NETWORK
TITLE =ML_LABORFREIGABE_T6
// Act 031
// Box           : LT-CIP
// Output address: Q258.5
      CALL FC    70 (
           UnitNo                   := #UnitNo,
           ActRec                   := DB2060.ML_LABORFREIGABE_T6,
           Typ                      := 0,
           FBa                      := #xTmp,
           FBa2                     := #xTmp,
           Out                      := Q    258.5);

END_FUNCTION_BLOCK

FUNCTION_BLOCK FB 1061
TITLE =U006: Water Tank 6
FAMILY : BOTEC_F1
NAME : UniE
VERSION : 1.2


VAR_TEMP
  CIP : BOOL ;	//CIP active
  UNIM : BOOL ;	//Unit Not In Maintenance
  GenRel : BOOL ;	//general OK (emergency and maintenance OK)
  EStopOK : BOOL ;	//emergency OK
  UnitNo : INT ;	//unit number
  xTmp : BOOL ;	//Temporary Bool
  iTmp : INT ;	//Temporary INT
  rTmp : REAL ;	//Temporary REAL
  dTmp : DINT ;	//Temporary DINT (free for general use)
  RetValInt : INT ;	//return value
END_VAR
BEGIN
NETWORK
TITLE =General

      SET   ;
// Simulation ---------------------------------------------------------------
      A     DB1061.DBX 1357.7;
      CC    FB  1069; // "WT06Sim"
      A     DB1061.DBX   17.3;
      =     DB1061.DBX 1357.7; //Help bit for simulation

// get unit number ----------------------------------------------------------
      L     DB1060.DBW    0;
      T     #UnitNo;

// communication ------------------------------------------------------------
      UC    FB  1065; // WT06Com

NETWORK
TITLE =Sequence organisation

      CLR   ;
      =     M    122.2;

// CIP Counter
      CALL FC    29 (
           UnitNo                   := #UnitNo,
           Value                    := DB1065.DBD   54,
           Enable                   := TRUE,
           Down                     := FALSE,
           OriginDetect             := 0.000000e+000,
           MaxDiffPS                := 1.000000e+000,
           SFMRec                   := DB1061.Seq.SFM[15],
           ValueOld                 := DB1061.DBD 1418);

// sequencer ----------------------------------------------------------------
      A     DB1063.DBX   43.1;
      S     DB1063.DBX   97.3;

      CALL FC    40 (
           UnitNo                   := #UnitNo);

END_FUNCTION_BLOCK

FUNCTION_BLOCK FB 1070
TITLE =U007: Wassertank 07
FAMILY : BOTEC_F1
NAME : U007A
VERSION : 2.1


VAR_TEMP
  EStopOK : BOOL ;	//auxiliary flag
  CIP : BOOL ;	//CIP Program Selected
  xTmp : BOOL ;	//Temporary Bool(free for general use)
  DummyBool : BOOL ;	//Temporary Bool(free for general use)
  UnitNo : INT ;	//unit number
  UnitFB : INT ;	//unit expansion FB number
  rTmp : REAL ;	//Temporary REAL (free for general use)
  iTmp : INT ;	//Temporary INT (free for general use)
  DummyInt : INT ;	//Temporary INT (free for general use)
  dTmp : DINT ;	//Temporary DINT (free for general use)
END_VAR
BEGIN
NETWORK
TITLE =general

      CLR   ;
      =     #xTmp;
      =     #EStopOK;

      L     DB1070.DBW    0;
      T     #UnitNo;
      L     DB1070.DBW    2;
      T     #UnitFB;

NETWORK
TITLE =analog inputs

      NOP   0;
// LI_T7 AnI 001 Inhalt Tank 7
      CALL FC    24 (
           UnitNo                   := #UnitNo,
           AnIRec                   := DB2073.LI_T7,
           ValPer                   := DB302.DBW   76);

NETWORK
TITLE =Universal value

      NOP   0;
// unv001 UnV 001 Process Status
      CALL FC    27 (
           UnitNo                   := #UnitNo,
           UnVRec                   := DB2075.unv001,
           ValExt                   := DB2075.DBD  234);

// unv002 UnV 002 Universal Value 02
      CALL FC    27 (
           UnitNo                   := #UnitNo,
           UnVRec                   := DB2075.unv002,
           ValExt                   := DB2075.DBD  362);

// unv003 UnV 003 Universal Value 03
      CALL FC    27 (
           UnitNo                   := #UnitNo,
           UnVRec                   := DB2075.unv003,
           ValExt                   := DB2075.DBD  490);

NETWORK
TITLE =special inputs

      NOP   0;
// LS_LLL_T7 SpI 001
      CALL FC    14 (
           UnitNo                   := #UnitNo,
           SpIRec                   := DB2071.LS_LLL_T7,
           SpIBit                   := I     71.0);

// LS_HL_T7 SpI 002
      CALL FC    14 (
           UnitNo                   := #UnitNo,
           SpIRec                   := DB2071.LS_HL_T7,
           SpIBit                   := I     70.6);

// LS_LL_T7 SpI 005
      CALL FC    14 (
           UnitNo                   := #UnitNo,
           SpIRec                   := DB2071.LS_LL_T7,
           SpIBit                   := I     70.7);

// RM_NI_T7_K2 SpI 008
      CALL FC    14 (
           UnitNo                   := #UnitNo,
           SpIRec                   := DB2071.RM_NI_T7_K2,
           SpIBit                   := I     61.2);

// RM_NI_T7_K3 SpI 010
      CALL FC    14 (
           UnitNo                   := #UnitNo,
           SpIRec                   := DB2071.RM_NI_T7_K3,
           SpIBit                   := I     69.4);

// LABOR_FREIG_T7 SpI 011 SCHLUESSELSCHALTER LABOR
      CALL FC    14 (
           UnitNo                   := #UnitNo,
           SpIRec                   := DB2071.LABOR_FREIG_T7,
           SpIBit                   := I    258.6);

NETWORK
TITLE =messages

      NOP   0;
// msg001 Msg 001 Message 01
      CALL FC    16 (
           UnitNo                   := #UnitNo,
           MsgRec                   := DB2077.msg001,
           MsgBit                   := DB2077.DBX   82.7);

// msg002 Msg 002 Message 02
      CALL FC    16 (
           UnitNo                   := #UnitNo,
           MsgRec                   := DB2077.msg002,
           MsgBit                   := DB2077.DBX  142.7);

NETWORK
TITLE =unit supply

      UC    FB [#UnitFB];

NETWORK
TITLE =T7_FW
// Act 001
// Box           : Ventilinsel 5
// Input address : I338.3
// Output address: Q338.3
      CALL FC    70 (
           UnitNo                   := #UnitNo,
           ActRec                   := DB2070.T7_FW,
           Typ                      := 1,
           FBa                      := #xTmp,
           FBa2                     := I    338.3,
           Out                      := Q    338.3);

NETWORK
TITLE =T7_KEG
// Act 003
// Box           : Ventilinsel 5
// Input address : I339.1
// Output address: Q339.1
      CALL FC    70 (
           UnitNo                   := #UnitNo,
           ActRec                   := DB2070.T7_KEG,
           Typ                      := 1,
           FBa                      := #xTmp,
           FBa2                     := I    339.1,
           Out                      := Q    339.1);

NETWORK
TITLE =T7_SK
// Act 004
// Box           : Ventilinsel 5
// Input address : I338.0
// Output address: Q338.0
      CALL FC    70 (
           UnitNo                   := #UnitNo,
           ActRec                   := DB2070.T7_SK,
           Typ                      := 1,
           FBa                      := #xTmp,
           FBa2                     := I    338.0,
           Out                      := Q    338.0);

NETWORK
TITLE =T7_A10
// Act 005
// Box           : Ventilinsel 2
// Input address : I316.2
// Output address: Q316.2
      CALL FC    70 (
           UnitNo                   := #UnitNo,
           ActRec                   := DB2070.T7_A10,
           Typ                      := 1,
           FBa                      := #xTmp,
           FBa2                     := I    316.2,
           Out                      := Q    316.2);

NETWORK
TITLE =T7_A9
// Act 006
// Box           : Ventilinsel 2
// Input address : I318.2
// Output address: Q318.2
      CALL FC    70 (
           UnitNo                   := #UnitNo,
           ActRec                   := DB2070.T7_A9,
           Typ                      := 1,
           FBa                      := #xTmp,
           FBa2                     := I    318.2,
           Out                      := Q    318.2);

NETWORK
TITLE =T7_A12
// Act 007
// Box           : Ventilinsel 2
// Input address : I320.2
// Output address: Q320.2
      CALL FC    70 (
           UnitNo                   := #UnitNo,
           ActRec                   := DB2070.T7_A12,
           Typ                      := 1,
           FBa                      := #xTmp,
           FBa2                     := I    320.2,
           Out                      := Q    320.2);

NETWORK
TITLE =T7_A7
// Act 008
// Box           : Ventilinsel 2
// Input address : I322.2
// Output address: Q322.2
      CALL FC    70 (
           UnitNo                   := #UnitNo,
           ActRec                   := DB2070.T7_A7,
           Typ                      := 1,
           FBa                      := #xTmp,
           FBa2                     := I    322.2,
           Out                      := Q    322.2);

NETWORK
TITLE =T7_A8
// Act 009
// Box           : Ventilinsel 3
// Input address : I324.2
// Output address: Q324.2
      CALL FC    70 (
           UnitNo                   := #UnitNo,
           ActRec                   := DB2070.T7_A8,
           Typ                      := 1,
           FBa                      := #xTmp,
           FBa2                     := I    324.2,
           Out                      := Q    324.2);

NETWORK
TITLE =T7_A5
// Act 010
// Box           : Ventilinsel 3
// Input address : I326.2
// Output address: Q326.2
      CALL FC    70 (
           UnitNo                   := #UnitNo,
           ActRec                   := DB2070.T7_A5,
           Typ                      := 1,
           FBa                      := #xTmp,
           FBa2                     := I    326.2,
           Out                      := Q    326.2);

NETWORK
TITLE =T7_A11
// Act 011
// Box           : Ventilinsel 3
// Input address : I328.2
// Output address: Q328.2
      CALL FC    70 (
           UnitNo                   := #UnitNo,
           ActRec                   := DB2070.T7_A11,
           Typ                      := 1,
           FBa                      := #xTmp,
           FBa2                     := I    328.2,
           Out                      := Q    328.2);

NETWORK
TITLE =T7_A14
// Act 012
// Box           : Ventilinsel 4
// Input address : I330.2
// Output address: Q330.2
      CALL FC    70 (
           UnitNo                   := #UnitNo,
           ActRec                   := DB2070.T7_A14,
           Typ                      := 1,
           FBa                      := #xTmp,
           FBa2                     := I    330.2,
           Out                      := Q    330.2);

NETWORK
TITLE =T7_A15
// Act 013
// Box           : Ventilinsel 4
// Input address : I332.2
// Output address: Q332.2
      CALL FC    70 (
           UnitNo                   := #UnitNo,
           ActRec                   := DB2070.T7_A15,
           Typ                      := 0,
           FBa                      := #xTmp,
           FBa2                     := I    332.2,
           Out                      := Q    332.2);

NETWORK
TITLE =T7_RR1
// Act 014
// Box           : Ventilinsel 4
// Input address : I334.2
// Output address: Q334.2
      CALL FC    70 (
           UnitNo                   := #UnitNo,
           ActRec                   := DB2070.T7_RR1,
           Typ                      := 1,
           FBa                      := #xTmp,
           FBa2                     := I    334.2,
           Out                      := Q    334.2);

NETWORK
TITLE =RV1_T7  RV1_T7 Ventil CIP Vorlauf Tank 7
// Act 015
// Box           : VS2-BB
// Input address : I304.1
// Output address: Q304.1
      CALL FC    70 (
           UnitNo                   := #UnitNo,
           ActRec                   := DB2070.RV1_T7,
           Typ                      := 1,
           FBa                      := #xTmp,
           FBa2                     := I    304.1,
           Out                      := Q    304.1);

NETWORK
TITLE =B6F_T7  B6F_T7
// Act 016
// Box           : VS2-BB
// Input address : I304.5
// Output address: Q304.5
      CALL FC    70 (
           UnitNo                   := #UnitNo,
           ActRec                   := DB2070.B6F_T7,
           Typ                      := 1,
           FBa                      := #xTmp,
           FBa2                     := I    304.5,
           Out                      := Q    304.5);

NETWORK
TITLE =H6F_T7  H6F_T7
// Act 017
// Box           : VS2-BB
// Input address : I304.4
// Output address: Q304.4
      CALL FC    70 (
           UnitNo                   := #UnitNo,
           ActRec                   := DB2070.H6F_T7,
           Typ                      := 1,
           FBa                      := #xTmp,
           FBa2                     := I    304.4,
           Out                      := Q    304.4);

NETWORK
TITLE =J6F_T7  J6F_T7
// Act 018
// Box           : VS2-BB
// Input address : I304.6
// Output address: Q304.6
      CALL FC    70 (
           UnitNo                   := #UnitNo,
           ActRec                   := DB2070.J6F_T7,
           Typ                      := 1,
           FBa                      := #xTmp,
           FBa2                     := I    304.6,
           Out                      := Q    304.6);

NETWORK
TITLE =L6F_T7  L6F_T7
// Act 019
// Box           : VS2-BB
// Input address : I304.7
// Output address: Q304.7
      CALL FC    70 (
           UnitNo                   := #UnitNo,
           ActRec                   := DB2070.L6F_T7,
           Typ                      := 1,
           FBa                      := #xTmp,
           FBa2                     := I    304.7,
           Out                      := Q    304.7);

NETWORK
TITLE =D6_T7  D6_T7
// Act 020
// Box           : VS2-BB
// Input address : I305.1
// Output address: Q305.1
      CALL FC    70 (
           UnitNo                   := #UnitNo,
           ActRec                   := DB2070.D6_T7,
           Typ                      := 1,
           FBa                      := #xTmp,
           FBa2                     := I    305.1,
           Out                      := Q    305.1);

NETWORK
TITLE =B6_T7  B6_T7
// Act 021
// Box           : VS2-BB
// Input address : I305.0
// Output address: Q305.0
      CALL FC    70 (
           UnitNo                   := #UnitNo,
           ActRec                   := DB2070.B6_T7,
           Typ                      := 1,
           FBa                      := #xTmp,
           FBa2                     := I    305.0,
           Out                      := Q    305.0);

NETWORK
TITLE =A_T7  A_T7
// Act 022
// Box           : VS2-BB
// Input address : I304.2
// Output address: Q304.2
      CALL FC    70 (
           UnitNo                   := #UnitNo,
           ActRec                   := DB2070.A_T7,
           Typ                      := 1,
           FBa                      := #xTmp,
           FBa2                     := I    304.2,
           Out                      := Q    304.2);

NETWORK
TITLE =B_T7  B_T7
// Act 023
// Box           : VS2-BB
// Input address : I304.3
// Output address: Q304.3
      CALL FC    70 (
           UnitNo                   := #UnitNo,
           ActRec                   := DB2070.B_T7,
           Typ                      := 1,
           FBa                      := #xTmp,
           FBa2                     := I    304.3,
           Out                      := Q    304.3);

NETWORK
TITLE =CF_T7
// Act 024
// Box           : Ventilinsel 1
// Input address : I17.0
// Output address: Q17.0
      CALL FC    70 (
           UnitNo                   := #UnitNo,
           ActRec                   := DB2070.CF_T7,
           Typ                      := 1,
           FBa                      := #xTmp,
           FBa2                     := I     17.0,
           Out                      := Q     17.0);

NETWORK
TITLE =RW5_T7  RW5_T7
// Act 026
// Box           : VS2-BB
// Input address : I305.2
// Output address: Q305.2
      CALL FC    70 (
           UnitNo                   := #UnitNo,
           ActRec                   := DB2070.RW5_T7,
           Typ                      := 1,
           FBa                      := #xTmp,
           FBa2                     := I    305.2,
           Out                      := Q    305.2);

NETWORK
TITLE =RW6_T7  RW6_T7
// Act 027
// Box           : VS2-BB
// Input address : I305.3
// Output address: Q305.3
      CALL FC    70 (
           UnitNo                   := #UnitNo,
           ActRec                   := DB2070.RW6_T7,
           Typ                      := 1,
           FBa                      := #xTmp,
           FBa2                     := I    305.3,
           Out                      := Q    305.3);

NETWORK
TITLE =VR_T7  VR_T7
// Act 029
// Box           : VS2-BB
// Output address: Q305.4
      CALL FC    70 (
           UnitNo                   := #UnitNo,
           ActRec                   := DB2070.VR_T7,
           Typ                      := 0,
           FBa                      := #xTmp,
           FBa2                     := #xTmp,
           Out                      := Q    305.4);

NETWORK
TITLE =ML_LABORFREIGABE_T7
// Act 031
// Box           : LT-CIP
// Output address: Q258.6
      CALL FC    70 (
           UnitNo                   := #UnitNo,
           ActRec                   := DB2070.ML_LABORFREIGABE_T7,
           Typ                      := 0,
           FBa                      := #xTmp,
           FBa2                     := #xTmp,
           Out                      := Q    258.6);

END_FUNCTION_BLOCK

FUNCTION_BLOCK FB 1071
TITLE =U007: Water Tank 7
FAMILY : BOTEC_F1
NAME : UniE
VERSION : 1.2


VAR_TEMP
  CIP : BOOL ;	//CIP active
  UNIM : BOOL ;	//Unit Not In Maintenance
  GenRel : BOOL ;	//general OK (emergency and maintenance OK)
  EStopOK : BOOL ;	//emergency OK
  UnitNo : INT ;	//unit number
  xTmp : BOOL ;	//Temporary Bool
  iTmp : INT ;	//Temporary INT
  rTmp : REAL ;	//Temporary REAL
  dTmp : DINT ;	//Temporary DINT (free for general use)
  RetValInt : INT ;	//return value
END_VAR
BEGIN
NETWORK
TITLE =General

      SET   ;
// Simulation ---------------------------------------------------------------
      A     DB1071.DBX 1357.7;
      CC    FB  1079; // "WT07Sim"
      A     DB1071.DBX   17.3;
      =     DB1071.DBX 1357.7; //Help bit for simulation

// get unit number ----------------------------------------------------------
      L     DB1070.DBW    0;
      T     #UnitNo;


// communication ------------------------------------------------------------
      UC    FB  1075; // WT07Com

NETWORK
TITLE =Sequence organisation

      CLR   ;
      =     M    122.2;

// CIP Counter
      CALL FC    29 (
           UnitNo                   := #UnitNo,
           Value                    := DB1075.DBD   54,
           Enable                   := TRUE,
           Down                     := FALSE,
           OriginDetect             := 0.000000e+000,
           MaxDiffPS                := 1.000000e+000,
           SFMRec                   := DB1071.Seq.SFM[15],
           ValueOld                 := DB1071.DBD 1418);

// sequencer ----------------------------------------------------------------
      A     DB1073.DBX   43.1;
      S     DB1073.DBX   97.3;

      CALL FC    40 (
           UnitNo                   := #UnitNo);

END_FUNCTION_BLOCK

FUNCTION_BLOCK FB 1080
TITLE =U008: Wassertank 08
FAMILY : BOTEC_F1
NAME : U008A
VERSION : 2.1


VAR_TEMP
  EStopOK : BOOL ;	//auxiliary flag
  CIP : BOOL ;	//CIP Program Selected
  xTmp : BOOL ;	//Temporary Bool(free for general use)
  DummyBool : BOOL ;	//Temporary Bool(free for general use)
  UnitNo : INT ;	//unit number
  UnitFB : INT ;	//unit expansion FB number
  rTmp : REAL ;	//Temporary REAL (free for general use)
  iTmp : INT ;	//Temporary INT (free for general use)
  DummyInt : INT ;	//Temporary INT (free for general use)
  dTmp : DINT ;	//Temporary DINT (free for general use)
END_VAR
BEGIN
NETWORK
TITLE =general

      CLR   ;
      =     #xTmp;
      =     #EStopOK;

      L     DB1080.DBW    0;
      T     #UnitNo;
      L     DB1080.DBW    2;
      T     #UnitFB;

NETWORK
TITLE =analog inputs

      NOP   0;
// LI_T8 AnI 001 Inhalt Tank 8
      CALL FC    24 (
           UnitNo                   := #UnitNo,
           AnIRec                   := DB2083.LI_T8,
           ValPer                   := DB302.DBW   78);

NETWORK
TITLE =Universal value

      NOP   0;
// unv001 UnV 001 Process Status
      CALL FC    27 (
           UnitNo                   := #UnitNo,
           UnVRec                   := DB2085.unv001,
           ValExt                   := DB2085.DBD  234);

// unv002 UnV 002 Universal Value 02
      CALL FC    27 (
           UnitNo                   := #UnitNo,
           UnVRec                   := DB2085.unv002,
           ValExt                   := DB2085.DBD  362);

// unv003 UnV 003 Universal Value 03
      CALL FC    27 (
           UnitNo                   := #UnitNo,
           UnVRec                   := DB2085.unv003,
           ValExt                   := DB2085.DBD  490);

NETWORK
TITLE =special inputs

      NOP   0;
// LS_LLL_T8 SpI 001
      CALL FC    14 (
           UnitNo                   := #UnitNo,
           SpIRec                   := DB2081.LS_LLL_T8,
           SpIBit                   := I    184.7);

// LS_HL_T8 SpI 002
      CALL FC    14 (
           UnitNo                   := #UnitNo,
           SpIRec                   := DB2081.LS_HL_T8,
           SpIBit                   := I    184.5);

// RM_NI_T8_ML SpI 003
      CALL FC    14 (
           UnitNo                   := #UnitNo,
           SpIRec                   := DB2081.RM_NI_T8_ML,
           SpIBit                   := I    184.4);

// RM_NI_T8_VV SpI 004 RM Vacuumventil Tank 8 ZU=1
      CALL FC    14 (
           UnitNo                   := #UnitNo,
           SpIRec                   := DB2081.RM_NI_T8_VV,
           SpIBit                   := I    184.6);

// LS_LL_T8 SpI 005
      CALL FC    14 (
           UnitNo                   := #UnitNo,
           SpIRec                   := DB2081.LS_LL_T8,
           SpIBit                   := I    185.7);

// RM_NI_T8_K4_AUF SpI 006 RM Klappe vor Filter Tank 8 AUF=1
      CALL FC    14 (
           UnitNo                   := #UnitNo,
           SpIRec                   := DB2081.RM_NI_T8_K4_AUF,
           SpIBit                   := I    186.1);

// RM_NI_T8_K4_ZU SpI 007 RM Klappe vor Filter Tank 8 ZU=1
      CALL FC    14 (
           UnitNo                   := #UnitNo,
           SpIRec                   := DB2081.RM_NI_T8_K4_ZU,
           SpIBit                   := I    184.3);

// RM_NI_T8_K2 SpI 008
      CALL FC    14 (
           UnitNo                   := #UnitNo,
           SpIRec                   := DB2081.RM_NI_T8_K2,
           SpIBit                   := I    184.1);

// RM_NI_T8_K3 SpI 010
      CALL FC    14 (
           UnitNo                   := #UnitNo,
           SpIRec                   := DB2081.RM_NI_T8_K3,
           SpIBit                   := I    184.2);

// LABOR_FREIG_T8 SpI 011 SCHLUESSELSCHALTER LABOR
      CALL FC    14 (
           UnitNo                   := #UnitNo,
           SpIRec                   := DB2081.LABOR_FREIG_T8,
           SpIBit                   := I    259.0);

NETWORK
TITLE =messages

      NOP   0;
// msg001 Msg 001 Message 01
      CALL FC    16 (
           UnitNo                   := #UnitNo,
           MsgRec                   := DB2087.msg001,
           MsgBit                   := DB2087.DBX   82.7);

// msg002 Msg 002 Message 02
      CALL FC    16 (
           UnitNo                   := #UnitNo,
           MsgRec                   := DB2087.msg002,
           MsgBit                   := DB2087.DBX  142.7);

NETWORK
TITLE =unit supply

      UC    FB [#UnitFB];

NETWORK
TITLE =T8_A10
// Act 005
// Box           : Ventilinsel 2
// Input address : I316.1
// Output address: Q316.1
      CALL FC    70 (
           UnitNo                   := #UnitNo,
           ActRec                   := DB2080.T8_A10,
           Typ                      := 1,
           FBa                      := #xTmp,
           FBa2                     := I    316.1,
           Out                      := Q    316.1);

NETWORK
TITLE =T8_A9
// Act 006
// Box           : Ventilinsel 2
// Input address : I318.1
// Output address: Q318.1
      CALL FC    70 (
           UnitNo                   := #UnitNo,
           ActRec                   := DB2080.T8_A9,
           Typ                      := 1,
           FBa                      := #xTmp,
           FBa2                     := I    318.1,
           Out                      := Q    318.1);

NETWORK
TITLE =T8_A12
// Act 007
// Box           : Ventilinsel 2
// Input address : I320.1
// Output address: Q320.1
      CALL FC    70 (
           UnitNo                   := #UnitNo,
           ActRec                   := DB2080.T8_A12,
           Typ                      := 1,
           FBa                      := #xTmp,
           FBa2                     := I    320.1,
           Out                      := Q    320.1);

NETWORK
TITLE =T8_A7
// Act 008
// Box           : Ventilinsel 2
// Input address : I322.1
// Output address: Q322.1
      CALL FC    70 (
           UnitNo                   := #UnitNo,
           ActRec                   := DB2080.T8_A7,
           Typ                      := 1,
           FBa                      := #xTmp,
           FBa2                     := I    322.1,
           Out                      := Q    322.1);

NETWORK
TITLE =T8_A8
// Act 009
// Box           : Ventilinsel 3
// Input address : I324.1
// Output address: Q324.1
      CALL FC    70 (
           UnitNo                   := #UnitNo,
           ActRec                   := DB2080.T8_A8,
           Typ                      := 1,
           FBa                      := #xTmp,
           FBa2                     := I    324.1,
           Out                      := Q    324.1);

NETWORK
TITLE =T8_A5
// Act 010
// Box           : Ventilinsel 3
// Input address : I326.1
// Output address: Q326.1
      CALL FC    70 (
           UnitNo                   := #UnitNo,
           ActRec                   := DB2080.T8_A5,
           Typ                      := 1,
           FBa                      := #xTmp,
           FBa2                     := I    326.1,
           Out                      := Q    326.1);

NETWORK
TITLE =T8_A11
// Act 011
// Box           : Ventilinsel 3
// Input address : I328.1
// Output address: Q328.1
      CALL FC    70 (
           UnitNo                   := #UnitNo,
           ActRec                   := DB2080.T8_A11,
           Typ                      := 1,
           FBa                      := #xTmp,
           FBa2                     := I    328.1,
           Out                      := Q    328.1);

NETWORK
TITLE =T8_A14
// Act 012
// Box           : Ventilinsel 4
// Input address : I330.1
// Output address: Q330.1
      CALL FC    70 (
           UnitNo                   := #UnitNo,
           ActRec                   := DB2080.T8_A14,
           Typ                      := 1,
           FBa                      := #xTmp,
           FBa2                     := I    330.1,
           Out                      := Q    330.1);

NETWORK
TITLE =T8_A15
// Act 013
// Box           : Ventilinsel 4
// Input address : I332.1
// Output address: Q332.1
      CALL FC    70 (
           UnitNo                   := #UnitNo,
           ActRec                   := DB2080.T8_A15,
           Typ                      := 0,
           FBa                      := #xTmp,
           FBa2                     := I    332.1,
           Out                      := Q    332.1);

NETWORK
TITLE =T8_RR1
// Act 014
// Box           : Ventilinsel 4
// Input address : I334.1
// Output address: Q334.1
      CALL FC    70 (
           UnitNo                   := #UnitNo,
           ActRec                   := DB2080.T8_RR1,
           Typ                      := 1,
           FBa                      := #xTmp,
           FBa2                     := I    334.1,
           Out                      := Q    334.1);

NETWORK
TITLE =RV1_T8  RV1_T8
// Act 015
// Box           : VS2-BB
// Input address : I305.5
// Output address: Q305.5
      CALL FC    70 (
           UnitNo                   := #UnitNo,
           ActRec                   := DB2080.RV1_T8,
           Typ                      := 1,
           FBa                      := #xTmp,
           FBa2                     := I    305.5,
           Out                      := Q    305.5);

NETWORK
TITLE =B6F_T8  B6F_T8
// Act 016
// Box           : VS2-BB
// Input address : I306.1
// Output address: Q306.1
      CALL FC    70 (
           UnitNo                   := #UnitNo,
           ActRec                   := DB2080.B6F_T8,
           Typ                      := 1,
           FBa                      := #xTmp,
           FBa2                     := I    306.1,
           Out                      := Q    306.1);

NETWORK
TITLE =H6F_T8  H6F_T8
// Act 017
// Box           : VS2-BB
// Input address : I306.0
// Output address: Q306.0
      CALL FC    70 (
           UnitNo                   := #UnitNo,
           ActRec                   := DB2080.H6F_T8,
           Typ                      := 1,
           FBa                      := #xTmp,
           FBa2                     := I    306.0,
           Out                      := Q    306.0);

NETWORK
TITLE =J6F_T8  J6F_T8
// Act 018
// Box           : VS2-BB
// Input address : I306.2
// Output address: Q306.2
      CALL FC    70 (
           UnitNo                   := #UnitNo,
           ActRec                   := DB2080.J6F_T8,
           Typ                      := 1,
           FBa                      := #xTmp,
           FBa2                     := I    306.2,
           Out                      := Q    306.2);

NETWORK
TITLE =L6F_T8  L6F_T8
// Act 019
// Box           : VS2-BB
// Input address : I306.3
// Output address: Q306.3
      CALL FC    70 (
           UnitNo                   := #UnitNo,
           ActRec                   := DB2080.L6F_T8,
           Typ                      := 1,
           FBa                      := #xTmp,
           FBa2                     := I    306.3,
           Out                      := Q    306.3);

NETWORK
TITLE =D6_T8  D6_T8
// Act 020
// Box           : VS2-BB
// Input address : I306.5
// Output address: Q306.5
      CALL FC    70 (
           UnitNo                   := #UnitNo,
           ActRec                   := DB2080.D6_T8,
           Typ                      := 1,
           FBa                      := #xTmp,
           FBa2                     := I    306.5,
           Out                      := Q    306.5);

NETWORK
TITLE =B6_T8  B6_T8
// Act 021
// Box           : VS2-BB
// Input address : I306.4
// Output address: Q306.4
      CALL FC    70 (
           UnitNo                   := #UnitNo,
           ActRec                   := DB2080.B6_T8,
           Typ                      := 1,
           FBa                      := #xTmp,
           FBa2                     := I    306.4,
           Out                      := Q    306.4);

NETWORK
TITLE =A_T8  A_T8
// Act 022
// Box           : VS2-BB
// Input address : I305.6
// Output address: Q305.6
      CALL FC    70 (
           UnitNo                   := #UnitNo,
           ActRec                   := DB2080.A_T8,
           Typ                      := 1,
           FBa                      := #xTmp,
           FBa2                     := I    305.6,
           Out                      := Q    305.6);

NETWORK
TITLE =B_T8  B_T8
// Act 023
// Box           : VS2-BB
// Input address : I305.7
// Output address: Q305.7
      CALL FC    70 (
           UnitNo                   := #UnitNo,
           ActRec                   := DB2080.B_T8,
           Typ                      := 1,
           FBa                      := #xTmp,
           FBa2                     := I    305.7,
           Out                      := Q    305.7);

NETWORK
TITLE =CF_T8
// Act 024
// Box           : Ventilinsel 1
// Input address : I17.1
// Output address: Q17.1
      CALL FC    70 (
           UnitNo                   := #UnitNo,
           ActRec                   := DB2080.CF_T8,
           Typ                      := 1,
           FBa                      := #xTmp,
           FBa2                     := I     17.1,
           Out                      := Q     17.1);

NETWORK
TITLE =C_T8
// Act 025
// Box           : VS2-BB
// Input address : I311.2
// Output address: Q311.2
      CALL FC    70 (
           UnitNo                   := #UnitNo,
           ActRec                   := DB2080.C_T8,
           Typ                      := 1,
           FBa                      := #xTmp,
           FBa2                     := I    311.2,
           Out                      := Q    311.2);

NETWORK
TITLE =VR_T8  VR_T8
// Act 029
// Box           : VS2-BB
// Output address: Q306.6
      CALL FC    70 (
           UnitNo                   := #UnitNo,
           ActRec                   := DB2080.VR_T8,
           Typ                      := 0,
           FBa                      := #xTmp,
           FBa2                     := #xTmp,
           Out                      := Q    306.6);

NETWORK
TITLE =ML_LABORFREIGABE_T8
// Act 031
// Box           : LT-CIP
// Output address: Q259.0
      CALL FC    70 (
           UnitNo                   := #UnitNo,
           ActRec                   := DB2080.ML_LABORFREIGABE_T8,
           Typ                      := 0,
           FBa                      := #xTmp,
           FBa2                     := #xTmp,
           Out                      := Q    259.0);

END_FUNCTION_BLOCK

FUNCTION_BLOCK FB 1081
TITLE =U008: Water Tank 8
FAMILY : BOTEC_F1
NAME : UniE
VERSION : 1.2


VAR_TEMP
  CIP : BOOL ;	//CIP active
  UNIM : BOOL ;	//Unit Not In Maintenance
  GenRel : BOOL ;	//general OK (emergency and maintenance OK)
  EStopOK : BOOL ;	//emergency OK
  UnitNo : INT ;	//unit number
  xTmp : BOOL ;	//Temporary Bool
  iTmp : INT ;	//Temporary INT
  rTmp : REAL ;	//Temporary REAL
  dTmp : DINT ;	//Temporary DINT (free for general use)
  RetValInt : INT ;	//return value
END_VAR
BEGIN
NETWORK
TITLE =General

      SET   ;
// Simulation ---------------------------------------------------------------
      A     DB1081.DBX 1357.7;
      CC    FB  1089; // "WT08Sim"
      A     DB1081.DBX   17.3;
      =     DB1081.DBX 1357.7; //Help bit for simulation

// get unit number ----------------------------------------------------------
      L     DB1080.DBW    0;
      T     #UnitNo;

// communication ------------------------------------------------------------
      UC    FB  1085; // WT08Com

NETWORK
TITLE =Sequence organisation

      CLR   ;
      =     M    122.2;

// CIP Counter
      CALL FC    29 (
           UnitNo                   := #UnitNo,
           Value                    := DB1085.DBD   54,
           Enable                   := TRUE,
           Down                     := FALSE,
           OriginDetect             := 0.000000e+000,
           MaxDiffPS                := 1.000000e+000,
           SFMRec                   := DB1081.Seq.SFM[15],
           ValueOld                 := DB1081.DBD 1418);

// sequencer ----------------------------------------------------------------
      A     DB1083.DBX   43.1;
      S     DB1083.DBX   97.3;

      CALL FC    40 (
           UnitNo                   := #UnitNo);

END_FUNCTION_BLOCK

FUNCTION_BLOCK FB 1090
TITLE =U009: Wassertank 09
FAMILY : BOTEC_F1
NAME : U009A
VERSION : 2.1


VAR_TEMP
  EStopOK : BOOL ;	//auxiliary flag
  CIP : BOOL ;	//CIP Program Selected
  xTmp : BOOL ;	//Temporary Bool(free for general use)
  DummyBool : BOOL ;	//Temporary Bool(free for general use)
  UnitNo : INT ;	//unit number
  UnitFB : INT ;	//unit expansion FB number
  rTmp : REAL ;	//Temporary REAL (free for general use)
  iTmp : INT ;	//Temporary INT (free for general use)
  DummyInt : INT ;	//Temporary INT (free for general use)
  dTmp : DINT ;	//Temporary DINT (free for general use)
END_VAR
BEGIN
NETWORK
TITLE =general

      CLR   ;
      =     #xTmp;
      =     #EStopOK;

      L     DB1090.DBW    0;
      T     #UnitNo;
      L     DB1090.DBW    2;
      T     #UnitFB;

NETWORK
TITLE =analog inputs

      NOP   0;
// LI_T9 AnI 001 Inhalt Tank 9
      CALL FC    24 (
           UnitNo                   := #UnitNo,
           AnIRec                   := DB2093.LI_T9,
           ValPer                   := DB302.DBW   80);

NETWORK
TITLE =Universal value

      NOP   0;
// unv001 UnV 001 Process Status
      CALL FC    27 (
           UnitNo                   := #UnitNo,
           UnVRec                   := DB2095.unv001,
           ValExt                   := DB2095.DBD  234);

// unv002 UnV 002 Universal Value 02
      CALL FC    27 (
           UnitNo                   := #UnitNo,
           UnVRec                   := DB2095.unv002,
           ValExt                   := DB2095.DBD  362);

// unv003 UnV 003 Universal Value 03
      CALL FC    27 (
           UnitNo                   := #UnitNo,
           UnVRec                   := DB2095.unv003,
           ValExt                   := DB2095.DBD  490);

NETWORK
TITLE =special inputs

      NOP   0;
// LS_LLL_T9 SpI 001
      CALL FC    14 (
           UnitNo                   := #UnitNo,
           SpIRec                   := DB2091.LS_LLL_T9,
           SpIBit                   := I    185.6);

// LS_HL_T9 SpI 002
      CALL FC    14 (
           UnitNo                   := #UnitNo,
           SpIRec                   := DB2091.LS_HL_T9,
           SpIBit                   := I    185.4);

// RM_NI_T9_ML SpI 003
      CALL FC    14 (
           UnitNo                   := #UnitNo,
           SpIRec                   := DB2091.RM_NI_T9_ML,
           SpIBit                   := I    185.3);

// RM_NI_T9_VV SpI 004 RM Vacuumventil Tank 9 ZU=1
      CALL FC    14 (
           UnitNo                   := #UnitNo,
           SpIRec                   := DB2091.RM_NI_T9_VV,
           SpIBit                   := I    185.5);

// LS_LL_T9 SpI 005
      CALL FC    14 (
           UnitNo                   := #UnitNo,
           SpIRec                   := DB2091.LS_LL_T9,
           SpIBit                   := I    186.0);

// RM_NI_T9_K4_AUF SpI 006 RM Klappe vor Filter Tank 9 AUF=1
      CALL FC    14 (
           UnitNo                   := #UnitNo,
           SpIRec                   := DB2091.RM_NI_T9_K4_AUF,
           SpIBit                   := I    186.2);

// RM_NI_T9_K4_ZU SpI 007 RM Klappe vor Filter Tank 9 ZU=1
      CALL FC    14 (
           UnitNo                   := #UnitNo,
           SpIRec                   := DB2091.RM_NI_T9_K4_ZU,
           SpIBit                   := I    185.2);

// RM_NI_T9_K2 SpI 008
      CALL FC    14 (
           UnitNo                   := #UnitNo,
           SpIRec                   := DB2091.RM_NI_T9_K2,
           SpIBit                   := I    185.0);

// RM_NI_T9_K3 SpI 010
      CALL FC    14 (
           UnitNo                   := #UnitNo,
           SpIRec                   := DB2091.RM_NI_T9_K3,
           SpIBit                   := I    185.1);

// LABOR_FREIG_T9 SpI 011 SCHLUESSELSCHALTER LABOR
      CALL FC    14 (
           UnitNo                   := #UnitNo,
           SpIRec                   := DB2091.LABOR_FREIG_T9,
           SpIBit                   := I    259.1);

NETWORK
TITLE =messages

      NOP   0;
// msg001 Msg 001 Message 01
      CALL FC    16 (
           UnitNo                   := #UnitNo,
           MsgRec                   := DB2097.msg001,
           MsgBit                   := DB2097.DBX   82.7);

// msg002 Msg 002 Message 02
      CALL FC    16 (
           UnitNo                   := #UnitNo,
           MsgRec                   := DB2097.msg002,
           MsgBit                   := DB2097.DBX  142.7);

NETWORK
TITLE =unit supply

      UC    FB [#UnitFB];

NETWORK
TITLE =T9_A10
// Act 005
// Box           : Ventilinsel 2
// Input address : I316.0
// Output address: Q316.0
      CALL FC    70 (
           UnitNo                   := #UnitNo,
           ActRec                   := DB2090.T9_A10,
           Typ                      := 1,
           FBa                      := #xTmp,
           FBa2                     := I    316.0,
           Out                      := Q    316.0);

NETWORK
TITLE =T9_A9
// Act 006
// Box           : Ventilinsel 2
// Input address : I318.0
// Output address: Q318.0
      CALL FC    70 (
           UnitNo                   := #UnitNo,
           ActRec                   := DB2090.T9_A9,
           Typ                      := 1,
           FBa                      := #xTmp,
           FBa2                     := I    318.0,
           Out                      := Q    318.0);

NETWORK
TITLE =T9_A12
// Act 007
// Box           : Ventilinsel 2
// Input address : I320.0
// Output address: Q320.0
      CALL FC    70 (
           UnitNo                   := #UnitNo,
           ActRec                   := DB2090.T9_A12,
           Typ                      := 1,
           FBa                      := #xTmp,
           FBa2                     := I    320.0,
           Out                      := Q    320.0);

NETWORK
TITLE =T9_A7
// Act 008
// Box           : Ventilinsel 2
// Input address : I322.0
// Output address: Q322.0
      CALL FC    70 (
           UnitNo                   := #UnitNo,
           ActRec                   := DB2090.T9_A7,
           Typ                      := 1,
           FBa                      := #xTmp,
           FBa2                     := I    322.0,
           Out                      := Q    322.0);

NETWORK
TITLE =T9_A8
// Act 009
// Box           : Ventilinsel 3
// Input address : I324.0
// Output address: Q324.0
      CALL FC    70 (
           UnitNo                   := #UnitNo,
           ActRec                   := DB2090.T9_A8,
           Typ                      := 1,
           FBa                      := #xTmp,
           FBa2                     := I    324.0,
           Out                      := Q    324.0);

NETWORK
TITLE =T9_A5
// Act 010
// Box           : Ventilinsel 3
// Input address : I326.0
// Output address: Q326.0
      CALL FC    70 (
           UnitNo                   := #UnitNo,
           ActRec                   := DB2090.T9_A5,
           Typ                      := 1,
           FBa                      := #xTmp,
           FBa2                     := I    326.0,
           Out                      := Q    326.0);

NETWORK
TITLE =T9_A11
// Act 011
// Box           : Ventilinsel 3
// Input address : I328.0
// Output address: Q328.0
      CALL FC    70 (
           UnitNo                   := #UnitNo,
           ActRec                   := DB2090.T9_A11,
           Typ                      := 1,
           FBa                      := #xTmp,
           FBa2                     := I    328.0,
           Out                      := Q    328.0);

NETWORK
TITLE =T9_A14
// Act 012
// Box           : Ventilinsel 4
// Input address : I330.0
// Output address: Q330.0
      CALL FC    70 (
           UnitNo                   := #UnitNo,
           ActRec                   := DB2090.T9_A14,
           Typ                      := 1,
           FBa                      := #xTmp,
           FBa2                     := I    330.0,
           Out                      := Q    330.0);

NETWORK
TITLE =T9_A15
// Act 013
// Box           : Ventilinsel 4
// Input address : I332.0
// Output address: Q332.0
      CALL FC    70 (
           UnitNo                   := #UnitNo,
           ActRec                   := DB2090.T9_A15,
           Typ                      := 0,
           FBa                      := #xTmp,
           FBa2                     := I    332.0,
           Out                      := Q    332.0);

NETWORK
TITLE =T9_RR1
// Act 014
// Box           : Ventilinsel 4
// Input address : I334.0
// Output address: Q334.0
      CALL FC    70 (
           UnitNo                   := #UnitNo,
           ActRec                   := DB2090.T9_RR1,
           Typ                      := 1,
           FBa                      := #xTmp,
           FBa2                     := I    334.0,
           Out                      := Q    334.0);

NETWORK
TITLE =RV1_T9  RV1_T9
// Act 015
// Box           : VS2-BB
// Input address : I306.7
// Output address: Q306.7
      CALL FC    70 (
           UnitNo                   := #UnitNo,
           ActRec                   := DB2090.RV1_T9,
           Typ                      := 1,
           FBa                      := #xTmp,
           FBa2                     := I    306.7,
           Out                      := Q    306.7);

NETWORK
TITLE =B6F_T9  B6F_T9
// Act 016
// Box           : VS2-BB
// Input address : I307.3
// Output address: Q307.3
      CALL FC    70 (
           UnitNo                   := #UnitNo,
           ActRec                   := DB2090.B6F_T9,
           Typ                      := 1,
           FBa                      := #xTmp,
           FBa2                     := I    307.3,
           Out                      := Q    307.3);

NETWORK
TITLE =H6F_T9  H6F_T9
// Act 017
// Box           : VS2-BB
// Input address : I307.2
// Output address: Q307.2
      CALL FC    70 (
           UnitNo                   := #UnitNo,
           ActRec                   := DB2090.H6F_T9,
           Typ                      := 1,
           FBa                      := #xTmp,
           FBa2                     := I    307.2,
           Out                      := Q    307.2);

NETWORK
TITLE =J6F_T9  J6F_T9
// Act 018
// Box           : VS2-BB
// Input address : I307.4
// Output address: Q307.4
      CALL FC    70 (
           UnitNo                   := #UnitNo,
           ActRec                   := DB2090.J6F_T9,
           Typ                      := 1,
           FBa                      := #xTmp,
           FBa2                     := I    307.4,
           Out                      := Q    307.4);

NETWORK
TITLE =L6F_T9  L6F_T9
// Act 019
// Box           : VS2-BB
// Input address : I307.5
// Output address: Q307.5
      CALL FC    70 (
           UnitNo                   := #UnitNo,
           ActRec                   := DB2090.L6F_T9,
           Typ                      := 1,
           FBa                      := #xTmp,
           FBa2                     := I    307.5,
           Out                      := Q    307.5);

NETWORK
TITLE =D6_T9  D6_T9
// Act 020
// Box           : VS2-BB
// Input address : I307.7
// Output address: Q307.7
      CALL FC    70 (
           UnitNo                   := #UnitNo,
           ActRec                   := DB2090.D6_T9,
           Typ                      := 1,
           FBa                      := #xTmp,
           FBa2                     := I    307.7,
           Out                      := Q    307.7);

NETWORK
TITLE =B6_T9  B6_T9
// Act 021
// Box           : VS2-BB
// Input address : I307.6
// Output address: Q307.6
      CALL FC    70 (
           UnitNo                   := #UnitNo,
           ActRec                   := DB2090.B6_T9,
           Typ                      := 1,
           FBa                      := #xTmp,
           FBa2                     := I    307.6,
           Out                      := Q    307.6);

NETWORK
TITLE =A_T9  A_T9
// Act 022
// Box           : VS2-BB
// Input address : I307.0
// Output address: Q307.0
      CALL FC    70 (
           UnitNo                   := #UnitNo,
           ActRec                   := DB2090.A_T9,
           Typ                      := 1,
           FBa                      := #xTmp,
           FBa2                     := I    307.0,
           Out                      := Q    307.0);

NETWORK
TITLE =B_T9  B_T9
// Act 023
// Box           : VS2-BB
// Input address : I307.1
// Output address: Q307.1
      CALL FC    70 (
           UnitNo                   := #UnitNo,
           ActRec                   := DB2090.B_T9,
           Typ                      := 1,
           FBa                      := #xTmp,
           FBa2                     := I    307.1,
           Out                      := Q    307.1);

NETWORK
TITLE =CF_T9
// Act 024
// Box           : Ventilinsel 1
// Input address : I17.2
// Output address: Q17.2
      CALL FC    70 (
           UnitNo                   := #UnitNo,
           ActRec                   := DB2090.CF_T9,
           Typ                      := 1,
           FBa                      := #xTmp,
           FBa2                     := I     17.2,
           Out                      := Q     17.2);

NETWORK
TITLE =C_T9
// Act 025
// Box           : VS2-BB
// Input address : I311.3
// Output address: Q311.3
      CALL FC    70 (
           UnitNo                   := #UnitNo,
           ActRec                   := DB2090.C_T9,
           Typ                      := 1,
           FBa                      := #xTmp,
           FBa2                     := I    311.3,
           Out                      := Q    311.3);

NETWORK
TITLE =VR_T9  VR_T9
// Act 029
// Box           : VS2-BB
// Output address: Q308.0
      CALL FC    70 (
           UnitNo                   := #UnitNo,
           ActRec                   := DB2090.VR_T9,
           Typ                      := 0,
           FBa                      := #xTmp,
           FBa2                     := #xTmp,
           Out                      := Q    308.0);

NETWORK
TITLE =ML_LABORFREIGABE_T9
// Act 031
// Box           : LT-CIP
// Output address: Q259.1
      CALL FC    70 (
           UnitNo                   := #UnitNo,
           ActRec                   := DB2090.ML_LABORFREIGABE_T9,
           Typ                      := 0,
           FBa                      := #xTmp,
           FBa2                     := #xTmp,
           Out                      := Q    259.1);

END_FUNCTION_BLOCK

FUNCTION_BLOCK FB 1091
TITLE =U009: Water Tank 9
FAMILY : BOTEC_F1
NAME : UniE
VERSION : 1.2


VAR_TEMP
  CIP : BOOL ;	//CIP active
  UNIM : BOOL ;	//Unit Not In Maintenance
  GenRel : BOOL ;	//general OK (emergency and maintenance OK)
  EStopOK : BOOL ;	//emergency OK
  UnitNo : INT ;	//unit number
  xTmp : BOOL ;	//Temporary Bool
  iTmp : INT ;	//Temporary INT
  rTmp : REAL ;	//Temporary REAL
  dTmp : DINT ;	//Temporary DINT (free for general use)
  RetValInt : INT ;	//return value
END_VAR
BEGIN
NETWORK
TITLE =General

      SET   ;
// Simulation ---------------------------------------------------------------
      A     DB1091.DBX 1357.7;
      CC    FB  1099; // "WT09Sim"
      A     DB1091.DBX   17.3;
      =     DB1091.DBX 1357.7; //Help bit for simulation

// get unit number ----------------------------------------------------------
      L     DB1090.DBW    0;
      T     #UnitNo;

// communication ------------------------------------------------------------
      UC    FB  1095; // WT09Com

NETWORK
TITLE =Sequence organisation

      CLR   ;
      =     M    122.2;

// CIP Counter
      CALL FC    29 (
           UnitNo                   := #UnitNo,
           Value                    := DB1095.DBD   54,
           Enable                   := TRUE,
           Down                     := FALSE,
           OriginDetect             := 0.000000e+000,
           MaxDiffPS                := 1.000000e+000,
           SFMRec                   := DB1091.Seq.SFM[15],
           ValueOld                 := DB1091.DBD 1418);

// sequencer ----------------------------------------------------------------
      A     DB1093.DBX   43.1;
      S     DB1093.DBX   97.3;

      CALL FC    40 (
           UnitNo                   := #UnitNo);

END_FUNCTION_BLOCK

FUNCTION_BLOCK FB 1100
TITLE =U010: Wassertank 10
FAMILY : BOTEC_F1
NAME : U010A
VERSION : 2.1


VAR_TEMP
  EStopOK : BOOL ;	//auxiliary flag
  CIP : BOOL ;	//CIP Program Selected
  xTmp : BOOL ;	//Temporary Bool(free for general use)
  DummyBool : BOOL ;	//Temporary Bool(free for general use)
  UnitNo : INT ;	//unit number
  UnitFB : INT ;	//unit expansion FB number
  rTmp : REAL ;	//Temporary REAL (free for general use)
  iTmp : INT ;	//Temporary INT (free for general use)
  DummyInt : INT ;	//Temporary INT (free for general use)
  dTmp : DINT ;	//Temporary DINT (free for general use)
END_VAR
BEGIN
NETWORK
TITLE =general

      CLR   ;
      =     #xTmp;
      =     #EStopOK;

      L     DB1100.DBW    0;
      T     #UnitNo;
      L     DB1100.DBW    2;
      T     #UnitFB;

NETWORK
TITLE =analog inputs

      NOP   0;
// LI_T10 AnI 001 Niveau Tank 10
      CALL FC    24 (
           UnitNo                   := #UnitNo,
           AnIRec                   := DB2103.LI_T10,
           ValPer                   := DB302.DBW   82);

NETWORK
TITLE =Universal value

      NOP   0;
// unv001 UnV 001 Process Status
      CALL FC    27 (
           UnitNo                   := #UnitNo,
           UnVRec                   := DB2105.unv001,
           ValExt                   := DB2105.DBD  234);

// unv002 UnV 002 Universal Value 02
      CALL FC    27 (
           UnitNo                   := #UnitNo,
           UnVRec                   := DB2105.unv002,
           ValExt                   := DB2105.DBD  362);

// unv003 UnV 003 Universal Value 03
      CALL FC    27 (
           UnitNo                   := #UnitNo,
           UnVRec                   := DB2105.unv003,
           ValExt                   := DB2105.DBD  490);

NETWORK
TITLE =special inputs

      NOP   0;
// LS_LLL_T10 SpI 001 LS- Tank 10
      CALL FC    14 (
           UnitNo                   := #UnitNo,
           SpIRec                   := DB2101.LS_LLL_T10,
           SpIBit                   := I     51.1);

// LS_HL_T10 SpI 002 LS+ Tank 10
      CALL FC    14 (
           UnitNo                   := #UnitNo,
           SpIRec                   := DB2101.LS_HL_T10,
           SpIBit                   := I     50.7);

// GOA_T10_ML SpI 003 Mannloch Tank 10
      CALL FC    14 (
           UnitNo                   := #UnitNo,
           SpIRec                   := DB2101.GOA_T10_ML,
           SpIBit                   := I     50.6);

// GOA_VV_T10 SpI 004 Vacuumventil Tank 10
      CALL FC    14 (
           UnitNo                   := #UnitNo,
           SpIRec                   := DB2101.GOA_VV_T10,
           SpIBit                   := I     50.5);

// LS_LL_T10 SpI 005 LS/ Tank 10
      CALL FC    14 (
           UnitNo                   := #UnitNo,
           SpIRec                   := DB2101.LS_LL_T10,
           SpIBit                   := I     51.0);

// RM_NI_T10_K4_AUF SpI 006
      CALL FC    14 (
           UnitNo                   := #UnitNo,
           SpIRec                   := DB2101.RM_NI_T10_K4_AUF,
           SpIBit                   := I     50.3);

// RM_NI_T10_K4_ZU SpI 007
      CALL FC    14 (
           UnitNo                   := #UnitNo,
           SpIRec                   := DB2101.RM_NI_T10_K4_ZU,
           SpIBit                   := I     50.4);

// RM_NI_T10_K2 SpI 008
      CALL FC    14 (
           UnitNo                   := #UnitNo,
           SpIRec                   := DB2101.RM_NI_T10_K2,
           SpIBit                   := I     50.1);

// RM_NI_T10_K3 SpI 010
      CALL FC    14 (
           UnitNo                   := #UnitNo,
           SpIRec                   := DB2101.RM_NI_T10_K3,
           SpIBit                   := I     50.2);

// LABOR_FREIG_T10 SpI 011 SCHLUESSELSCHALTER LABOR
      CALL FC    14 (
           UnitNo                   := #UnitNo,
           SpIRec                   := DB2101.LABOR_FREIG_T10,
           SpIBit                   := I    259.2);

NETWORK
TITLE =messages

      NOP   0;
// msg001 Msg 001 Message 01
      CALL FC    16 (
           UnitNo                   := #UnitNo,
           MsgRec                   := DB2107.msg001,
           MsgBit                   := DB2107.DBX   82.7);

// msg002 Msg 002 Message 02
      CALL FC    16 (
           UnitNo                   := #UnitNo,
           MsgRec                   := DB2107.msg002,
           MsgBit                   := DB2107.DBX  142.7);

NETWORK
TITLE =unit supply

      UC    FB [#UnitFB];

NETWORK
TITLE =T10_A10
// Act 005
// Box           : Ventilinsel 2
// Input address : I317.1
// Output address: Q317.1
      CALL FC    70 (
           UnitNo                   := #UnitNo,
           ActRec                   := DB2100.T10_A10,
           Typ                      := 1,
           FBa                      := #xTmp,
           FBa2                     := I    317.1,
           Out                      := Q    317.1);

NETWORK
TITLE =T10_A9
// Act 006
// Box           : Ventilinsel 2
// Input address : I319.1
// Output address: Q319.1
      CALL FC    70 (
           UnitNo                   := #UnitNo,
           ActRec                   := DB2100.T10_A9,
           Typ                      := 1,
           FBa                      := #xTmp,
           FBa2                     := I    319.1,
           Out                      := Q    319.1);

NETWORK
TITLE =T10_A12
// Act 007
// Box           : Ventilinsel 2
// Input address : I321.1
// Output address: Q321.1
      CALL FC    70 (
           UnitNo                   := #UnitNo,
           ActRec                   := DB2100.T10_A12,
           Typ                      := 1,
           FBa                      := #xTmp,
           FBa2                     := I    321.1,
           Out                      := Q    321.1);

NETWORK
TITLE =T10_A7
// Act 008
// Box           : Ventilinsel 2
// Input address : I323.1
// Output address: Q323.1
      CALL FC    70 (
           UnitNo                   := #UnitNo,
           ActRec                   := DB2100.T10_A7,
           Typ                      := 1,
           FBa                      := #xTmp,
           FBa2                     := I    323.1,
           Out                      := Q    323.1);

NETWORK
TITLE =T10_A8
// Act 009
// Box           : Ventilinsel 3
// Input address : I325.1
// Output address: Q325.1
      CALL FC    70 (
           UnitNo                   := #UnitNo,
           ActRec                   := DB2100.T10_A8,
           Typ                      := 1,
           FBa                      := #xTmp,
           FBa2                     := I    325.1,
           Out                      := Q    325.1);

NETWORK
TITLE =T10_A5
// Act 010
// Box           : Ventilinsel 3
// Input address : I327.1
// Output address: Q327.1
      CALL FC    70 (
           UnitNo                   := #UnitNo,
           ActRec                   := DB2100.T10_A5,
           Typ                      := 1,
           FBa                      := #xTmp,
           FBa2                     := I    327.1,
           Out                      := Q    327.1);

NETWORK
TITLE =T10_A11
// Act 011
// Box           : Ventilinsel 3
// Input address : I329.1
// Output address: Q329.1
      CALL FC    70 (
           UnitNo                   := #UnitNo,
           ActRec                   := DB2100.T10_A11,
           Typ                      := 1,
           FBa                      := #xTmp,
           FBa2                     := I    329.1,
           Out                      := Q    329.1);

NETWORK
TITLE =T10_A14
// Act 012
// Box           : Ventilinsel 4
// Input address : I331.1
// Output address: Q331.1
      CALL FC    70 (
           UnitNo                   := #UnitNo,
           ActRec                   := DB2100.T10_A14,
           Typ                      := 1,
           FBa                      := #xTmp,
           FBa2                     := I    331.1,
           Out                      := Q    331.1);

NETWORK
TITLE =T10_A15
// Act 013
// Box           : Ventilinsel 4
// Input address : I333.1
// Output address: Q333.1
      CALL FC    70 (
           UnitNo                   := #UnitNo,
           ActRec                   := DB2100.T10_A15,
           Typ                      := 0,
           FBa                      := #xTmp,
           FBa2                     := I    333.1,
           Out                      := Q    333.1);

NETWORK
TITLE =T10_RR1
// Act 014
// Box           : Ventilinsel 4
// Input address : I335.1
// Output address: Q335.1
      CALL FC    70 (
           UnitNo                   := #UnitNo,
           ActRec                   := DB2100.T10_RR1,
           Typ                      := 1,
           FBa                      := #xTmp,
           FBa2                     := I    335.1,
           Out                      := Q    335.1);

NETWORK
TITLE =RV1_T10  RV1_T10
// Act 015
// Box           : VS2-BB
// Input address : I308.1
// Output address: Q308.1
      CALL FC    70 (
           UnitNo                   := #UnitNo,
           ActRec                   := DB2100.RV1_T10,
           Typ                      := 1,
           FBa                      := #xTmp,
           FBa2                     := I    308.1,
           Out                      := Q    308.1);

NETWORK
TITLE =B6F_T10  B6F_T10
// Act 016
// Box           : VS2-BB
// Input address : I308.5
// Output address: Q308.5
      CALL FC    70 (
           UnitNo                   := #UnitNo,
           ActRec                   := DB2100.B6F_T10,
           Typ                      := 1,
           FBa                      := #xTmp,
           FBa2                     := I    308.5,
           Out                      := Q    308.5);

NETWORK
TITLE =H6F_T10  H6F_T10
// Act 017
// Box           : VS2-BB
// Input address : I308.4
// Output address: Q308.4
      CALL FC    70 (
           UnitNo                   := #UnitNo,
           ActRec                   := DB2100.H6F_T10,
           Typ                      := 1,
           FBa                      := #xTmp,
           FBa2                     := I    308.4,
           Out                      := Q    308.4);

NETWORK
TITLE =J6F_T10  J6F_T10
// Act 018
// Box           : VS2-BB
// Input address : I308.6
// Output address: Q308.6
      CALL FC    70 (
           UnitNo                   := #UnitNo,
           ActRec                   := DB2100.J6F_T10,
           Typ                      := 1,
           FBa                      := #xTmp,
           FBa2                     := I    308.6,
           Out                      := Q    308.6);

NETWORK
TITLE =L6F_T10  L6F_T10
// Act 019
// Box           : VS2-BB
// Input address : I308.7
// Output address: Q308.7
      CALL FC    70 (
           UnitNo                   := #UnitNo,
           ActRec                   := DB2100.L6F_T10,
           Typ                      := 1,
           FBa                      := #xTmp,
           FBa2                     := I    308.7,
           Out                      := Q    308.7);

NETWORK
TITLE =D6_T10  D6_T10
// Act 020
// Box           : VS2-BB
// Input address : I309.1
// Output address: Q309.1
      CALL FC    70 (
           UnitNo                   := #UnitNo,
           ActRec                   := DB2100.D6_T10,
           Typ                      := 1,
           FBa                      := #xTmp,
           FBa2                     := I    309.1,
           Out                      := Q    309.1);

NETWORK
TITLE =B6_T10  B6_T10
// Act 021
// Box           : VS2-BB
// Input address : I309.0
// Output address: Q309.0
      CALL FC    70 (
           UnitNo                   := #UnitNo,
           ActRec                   := DB2100.B6_T10,
           Typ                      := 1,
           FBa                      := #xTmp,
           FBa2                     := I    309.0,
           Out                      := Q    309.0);

NETWORK
TITLE =A_T10  A_T10
// Act 022
// Box           : VS2-BB
// Input address : I308.2
// Output address: Q308.2
      CALL FC    70 (
           UnitNo                   := #UnitNo,
           ActRec                   := DB2100.A_T10,
           Typ                      := 1,
           FBa                      := #xTmp,
           FBa2                     := I    308.2,
           Out                      := Q    308.2);

NETWORK
TITLE =B_T10  B_T10
// Act 023
// Box           : VS2-BB
// Input address : I308.3
// Output address: Q308.3
      CALL FC    70 (
           UnitNo                   := #UnitNo,
           ActRec                   := DB2100.B_T10,
           Typ                      := 1,
           FBa                      := #xTmp,
           FBa2                     := I    308.3,
           Out                      := Q    308.3);

NETWORK
TITLE =CF_T10
// Act 024
// Box           : Ventilinsel 1
// Input address : I17.3
// Output address: Q17.3
//      CALL  "Act"
//       UnitNo:=#UnitNo
//       ActRec:="U010ActD".CF_T10
//       Typ   :=0
//       FBa   :=#xTmp
//       FBa2  :="CF_T10GSC"
//       Out   :="CF_T10O"

NETWORK
TITLE =VVT10   Vacuumventil Tank 10
// Act 028
// Box           :
// Input address : I50.5
// Output address: #DummyBool
      CALL FC    70 (
           UnitNo                   := #UnitNo,
           ActRec                   := DB2100.VVT10,
           Typ                      := 1,
           FBa                      := #xTmp,
           FBa2                     := I     50.5,
           Out                      := #DummyBool);

NETWORK
TITLE =VR_T10  VR_T10
// Act 029
// Box           : VS2-BB
// Output address: Q309.2
      CALL FC    70 (
           UnitNo                   := #UnitNo,
           ActRec                   := DB2100.VR_T10,
           Typ                      := 0,
           FBa                      := #xTmp,
           FBa2                     := #xTmp,
           Out                      := Q    309.2);

NETWORK
TITLE =ML_LABORFREIGABE_T10
// Act 031
// Box           : LT-CIP
// Output address: Q259.2
      CALL FC    70 (
           UnitNo                   := #UnitNo,
           ActRec                   := DB2100.ML_LABORFREIGABE_T10,
           Typ                      := 0,
           FBa                      := #xTmp,
           FBa2                     := #xTmp,
           Out                      := Q    259.2);

END_FUNCTION_BLOCK

FUNCTION_BLOCK FB 1101
TITLE =U010: Water Tank 10
FAMILY : BOTEC_F1
NAME : UniE
VERSION : 1.2


VAR_TEMP
  CIP : BOOL ;	//CIP active
  UNIM : BOOL ;	//Unit Not In Maintenance
  GenRel : BOOL ;	//general OK (emergency and maintenance OK)
  EStopOK : BOOL ;	//emergency OK
  UnitNo : INT ;	//unit number
  xTmp : BOOL ;	//Temporary Bool
  iTmp : INT ;	//Temporary INT
  rTmp : REAL ;	//Temporary REAL
  dTmp : DINT ;	//Temporary DINT (free for general use)
  RetValInt : INT ;	//return value
END_VAR
BEGIN
NETWORK
TITLE =General

      SET   ;
// Simulation ---------------------------------------------------------------
      A     DB1101.DBX 1357.7;
      CC    FB  1109; // "WT10Sim"
      A     DB1101.DBX   17.3;
      =     DB1101.DBX 1357.7; //Help bit for simulation

// get unit number ----------------------------------------------------------
      L     DB1100.DBW    0;
      T     #UnitNo;

// communication ------------------------------------------------------------
      UC    FB  1105; // WT10Com

NETWORK
TITLE =Sequence organisation

      CLR   ;
      =     M    122.2;

// CIP Counter
      CALL FC    29 (
           UnitNo                   := #UnitNo,
           Value                    := DB1105.DBD   54,
           Enable                   := TRUE,
           Down                     := FALSE,
           OriginDetect             := 0.000000e+000,
           MaxDiffPS                := 1.000000e+000,
           SFMRec                   := DB1101.Seq.SFM[15],
           ValueOld                 := DB1101.DBD 1418);

// sequencer ----------------------------------------------------------------
      A     DB1103.DBX   43.1;
      S     DB1103.DBX   97.3;

      CALL FC    40 (
           UnitNo                   := #UnitNo);

END_FUNCTION_BLOCK

FUNCTION_BLOCK FB 1110
TITLE =U011: Wassertank 11
FAMILY : BOTEC_F1
NAME : U011A
VERSION : 2.1


VAR_TEMP
  EStopOK : BOOL ;	//auxiliary flag
  CIP : BOOL ;	//CIP Program Selected
  xTmp : BOOL ;	//Temporary Bool(free for general use)
  DummyBool : BOOL ;	//Temporary Bool(free for general use)
  UnitNo : INT ;	//unit number
  UnitFB : INT ;	//unit expansion FB number
  rTmp : REAL ;	//Temporary REAL (free for general use)
  iTmp : INT ;	//Temporary INT (free for general use)
  DummyInt : INT ;	//Temporary INT (free for general use)
  dTmp : DINT ;	//Temporary DINT (free for general use)
END_VAR
BEGIN
NETWORK
TITLE =general

      CLR   ;
      =     #xTmp;
      =     #EStopOK;

      L     DB1110.DBW    0;
      T     #UnitNo;
      L     DB1110.DBW    2;
      T     #UnitFB;

NETWORK
TITLE =analog inputs

      NOP   0;
// LI_T11 AnI 001 Niveau Tank 11
      CALL FC    24 (
           UnitNo                   := #UnitNo,
           AnIRec                   := DB2113.LI_T11,
           ValPer                   := DB302.DBW   84);

NETWORK
TITLE =Universal value

      NOP   0;
// unv001 UnV 001 Process Status
      CALL FC    27 (
           UnitNo                   := #UnitNo,
           UnVRec                   := DB2115.unv001,
           ValExt                   := DB2115.DBD  234);

// unv002 UnV 002 Universal Value 02
      CALL FC    27 (
           UnitNo                   := #UnitNo,
           UnVRec                   := DB2115.unv002,
           ValExt                   := DB2115.DBD  362);

// unv003 UnV 003 Universal Value 03
      CALL FC    27 (
           UnitNo                   := #UnitNo,
           UnVRec                   := DB2115.unv003,
           ValExt                   := DB2115.DBD  490);

NETWORK
TITLE =special inputs

      NOP   0;
// LS_LLL_T11 SpI 001 LS- Tank 11
      CALL FC    14 (
           UnitNo                   := #UnitNo,
           SpIRec                   := DB2111.LS_LLL_T11,
           SpIBit                   := I    187.6);

// LS_HL_T11 SpI 002 LS+ Tank 11
      CALL FC    14 (
           UnitNo                   := #UnitNo,
           SpIRec                   := DB2111.LS_HL_T11,
           SpIBit                   := I    187.4);

// GOA_T11_ML SpI 003 Mannloch Tank 11
      CALL FC    14 (
           UnitNo                   := #UnitNo,
           SpIRec                   := DB2111.GOA_T11_ML,
           SpIBit                   := I    187.3);

// GOA_T11_VV SpI 004 Vacuumventil Tank 11
      CALL FC    14 (
           UnitNo                   := #UnitNo,
           SpIRec                   := DB2111.GOA_T11_VV,
           SpIBit                   := I    187.2);

// LS_LL_T11 SpI 005 LS/ Tank 11
      CALL FC    14 (
           UnitNo                   := #UnitNo,
           SpIRec                   := DB2111.LS_LL_T11,
           SpIBit                   := I    187.5);

// RM_NI_T11_K4_AUF SpI 006
      CALL FC    14 (
           UnitNo                   := #UnitNo,
           SpIRec                   := DB2111.RM_NI_T11_K4_AUF,
           SpIBit                   := I    187.0);

// RM_NI_T11_K4_ZU SpI 007
      CALL FC    14 (
           UnitNo                   := #UnitNo,
           SpIRec                   := DB2111.RM_NI_T11_K4_ZU,
           SpIBit                   := I    187.1);

// RM_NI_T11_K2 SpI 008
      CALL FC    14 (
           UnitNo                   := #UnitNo,
           SpIRec                   := DB2111.RM_NI_T11_K2,
           SpIBit                   := I    186.6);

// RM_NI_T11_K3 SpI 010
      CALL FC    14 (
           UnitNo                   := #UnitNo,
           SpIRec                   := DB2111.RM_NI_T11_K3,
           SpIBit                   := I    186.7);

// LABOR_FREIG_T11 SpI 011 SCHLUESSELSCHALTER LABOR
      CALL FC    14 (
           UnitNo                   := #UnitNo,
           SpIRec                   := DB2111.LABOR_FREIG_T11,
           SpIBit                   := I    259.3);

NETWORK
TITLE =messages

      NOP   0;
// msg001 Msg 001 Message 01
      CALL FC    16 (
           UnitNo                   := #UnitNo,
           MsgRec                   := DB2117.msg001,
           MsgBit                   := DB2117.DBX   82.7);

// msg002 Msg 002 Message 02
      CALL FC    16 (
           UnitNo                   := #UnitNo,
           MsgRec                   := DB2117.msg002,
           MsgBit                   := DB2117.DBX  142.7);

NETWORK
TITLE =unit supply

      UC    FB [#UnitFB];

NETWORK
TITLE =T11_A10
// Act 005
// Box           : Ventilinsel 2
// Input address : I317.2
// Output address: Q317.2
      CALL FC    70 (
           UnitNo                   := #UnitNo,
           ActRec                   := DB2110.T11_A10,
           Typ                      := 1,
           FBa                      := #xTmp,
           FBa2                     := I    317.2,
           Out                      := Q    317.2);

NETWORK
TITLE =T11_A9
// Act 006
// Box           : Ventilinsel 2
// Input address : I319.2
// Output address: Q319.2
      CALL FC    70 (
           UnitNo                   := #UnitNo,
           ActRec                   := DB2110.T11_A9,
           Typ                      := 1,
           FBa                      := #xTmp,
           FBa2                     := I    319.2,
           Out                      := Q    319.2);

NETWORK
TITLE =T11_A12
// Act 007
// Box           : Ventilinsel 2
// Input address : I321.2
// Output address: Q321.2
      CALL FC    70 (
           UnitNo                   := #UnitNo,
           ActRec                   := DB2110.T11_A12,
           Typ                      := 1,
           FBa                      := #xTmp,
           FBa2                     := I    321.2,
           Out                      := Q    321.2);

NETWORK
TITLE =T11_A7
// Act 008
// Box           : Ventilinsel 2
// Input address : I323.2
// Output address: Q323.2
      CALL FC    70 (
           UnitNo                   := #UnitNo,
           ActRec                   := DB2110.T11_A7,
           Typ                      := 1,
           FBa                      := #xTmp,
           FBa2                     := I    323.2,
           Out                      := Q    323.2);

NETWORK
TITLE =T11_A8
// Act 009
// Box           : Ventilinsel 3
// Input address : I325.2
// Output address: Q325.2
      CALL FC    70 (
           UnitNo                   := #UnitNo,
           ActRec                   := DB2110.T11_A8,
           Typ                      := 1,
           FBa                      := #xTmp,
           FBa2                     := I    325.2,
           Out                      := Q    325.2);

NETWORK
TITLE =T11_A5
// Act 010
// Box           : Ventilinsel 3
// Input address : I327.2
// Output address: Q327.2
      CALL FC    70 (
           UnitNo                   := #UnitNo,
           ActRec                   := DB2110.T11_A5,
           Typ                      := 1,
           FBa                      := #xTmp,
           FBa2                     := I    327.2,
           Out                      := Q    327.2);

NETWORK
TITLE =T11_A11
// Act 011
// Box           : Ventilinsel 3
// Input address : I329.2
// Output address: Q329.2
      CALL FC    70 (
           UnitNo                   := #UnitNo,
           ActRec                   := DB2110.T11_A11,
           Typ                      := 1,
           FBa                      := #xTmp,
           FBa2                     := I    329.2,
           Out                      := Q    329.2);

NETWORK
TITLE =T11_A14
// Act 012
// Box           : Ventilinsel 4
// Input address : I331.2
// Output address: Q331.2
      CALL FC    70 (
           UnitNo                   := #UnitNo,
           ActRec                   := DB2110.T11_A14,
           Typ                      := 1,
           FBa                      := #xTmp,
           FBa2                     := I    331.2,
           Out                      := Q    331.2);

NETWORK
TITLE =T11_A15
// Act 013
// Box           : Ventilinsel 4
// Input address : I333.2
// Output address: Q333.2
      CALL FC    70 (
           UnitNo                   := #UnitNo,
           ActRec                   := DB2110.T11_A15,
           Typ                      := 0,
           FBa                      := #xTmp,
           FBa2                     := I    333.2,
           Out                      := Q    333.2);

NETWORK
TITLE =T11_RR1
// Act 014
// Box           : Ventilinsel 4
// Input address : I335.2
// Output address: Q335.2
      CALL FC    70 (
           UnitNo                   := #UnitNo,
           ActRec                   := DB2110.T11_RR1,
           Typ                      := 1,
           FBa                      := #xTmp,
           FBa2                     := I    335.2,
           Out                      := Q    335.2);

NETWORK
TITLE =RV1_T11
// Act 015
// Box           : Ventilinsel 1
// Input address : I8.0
// Output address: Q8.0
      CALL FC    70 (
           UnitNo                   := #UnitNo,
           ActRec                   := DB2110.RV1_T11,
           Typ                      := 1,
           FBa                      := #xTmp,
           FBa2                     := I      8.0,
           Out                      := Q      8.0);

NETWORK
TITLE =B6F_T11
// Act 016
// Box           : Ventilinsel 1
// Input address : I8.1
// Output address: Q8.1
      CALL FC    70 (
           UnitNo                   := #UnitNo,
           ActRec                   := DB2110.B6F_T11,
           Typ                      := 1,
           FBa                      := #xTmp,
           FBa2                     := I      8.1,
           Out                      := Q      8.1);

NETWORK
TITLE =H6F_T11
// Act 017
// Box           : Ventilinsel 1
// Input address : I8.2
// Output address: Q8.2
      CALL FC    70 (
           UnitNo                   := #UnitNo,
           ActRec                   := DB2110.H6F_T11,
           Typ                      := 1,
           FBa                      := #xTmp,
           FBa2                     := I      8.2,
           Out                      := Q      8.2);

NETWORK
TITLE =J6F_T11
// Act 018
// Box           : Ventilinsel 1
// Input address : I8.3
// Output address: Q8.3
      CALL FC    70 (
           UnitNo                   := #UnitNo,
           ActRec                   := DB2110.J6F_T11,
           Typ                      := 1,
           FBa                      := #xTmp,
           FBa2                     := I      8.3,
           Out                      := Q      8.3);

NETWORK
TITLE =L6F_T11
// Act 019
// Box           : Ventilinsel 1
// Input address : I8.4
// Output address: Q8.4
      CALL FC    70 (
           UnitNo                   := #UnitNo,
           ActRec                   := DB2110.L6F_T11,
           Typ                      := 1,
           FBa                      := #xTmp,
           FBa2                     := I      8.4,
           Out                      := Q      8.4);

NETWORK
TITLE =D6_T11
// Act 020
// Box           : Ventilinsel 1
// Input address : I8.5
// Output address: Q8.5
      CALL FC    70 (
           UnitNo                   := #UnitNo,
           ActRec                   := DB2110.D6_T11,
           Typ                      := 1,
           FBa                      := #xTmp,
           FBa2                     := I      8.5,
           Out                      := Q      8.5);

NETWORK
TITLE =B6_T11
// Act 021
// Box           : Ventilinsel 1
// Input address : I8.6
// Output address: Q8.6
      CALL FC    70 (
           UnitNo                   := #UnitNo,
           ActRec                   := DB2110.B6_T11,
           Typ                      := 1,
           FBa                      := #xTmp,
           FBa2                     := I      8.6,
           Out                      := Q      8.6);

NETWORK
TITLE =A_T11
// Act 022
// Box           : Ventilinsel 1
// Input address : I8.7
// Output address: Q8.7
      CALL FC    70 (
           UnitNo                   := #UnitNo,
           ActRec                   := DB2110.A_T11,
           Typ                      := 1,
           FBa                      := #xTmp,
           FBa2                     := I      8.7,
           Out                      := Q      8.7);

NETWORK
TITLE =B_T11
// Act 023
// Box           : Ventilinsel 1
// Input address : I9.0
// Output address: Q9.0
      CALL FC    70 (
           UnitNo                   := #UnitNo,
           ActRec                   := DB2110.B_T11,
           Typ                      := 1,
           FBa                      := #xTmp,
           FBa2                     := I      9.0,
           Out                      := Q      9.0);

NETWORK
TITLE =CF_T11
// Act 024
// Box           : Ventilinsel 1
// Input address : I17.4
// Output address: Q17.4
      CALL FC    70 (
           UnitNo                   := #UnitNo,
           ActRec                   := DB2110.CF_T11,
           Typ                      := 1,
           FBa                      := #xTmp,
           FBa2                     := I     17.4,
           Out                      := Q     17.4);

NETWORK
TITLE =C_T11
// Act 025
// Box           : VS2-BB
// Input address : I311.4
// Output address: Q311.4
      CALL FC    70 (
           UnitNo                   := #UnitNo,
           ActRec                   := DB2110.C_T11,
           Typ                      := 1,
           FBa                      := #xTmp,
           FBa2                     := I    311.4,
           Out                      := Q    311.4);

NETWORK
TITLE =VVT11  Vacuumventil Tank 11
// Act 028
// Box           : VST1-9
// Output address: Q160.0
      CALL FC    70 (
           UnitNo                   := #UnitNo,
           ActRec                   := DB2110.VVT11,
           Typ                      := 0,
           FBa                      := #xTmp,
           FBa2                     := #xTmp,
           Out                      := Q    160.0);

NETWORK
TITLE =VR_T11
// Act 029
// Box           : Ventilinsel 1
// Output address: Q9.1
      CALL FC    70 (
           UnitNo                   := #UnitNo,
           ActRec                   := DB2110.VR_T11,
           Typ                      := 0,
           FBa                      := #xTmp,
           FBa2                     := #xTmp,
           Out                      := Q      9.1);

NETWORK
TITLE =ML_LABORFREIGABE_T11
// Act 031
// Box           : LT-CIP
// Output address: Q259.3
      CALL FC    70 (
           UnitNo                   := #UnitNo,
           ActRec                   := DB2110.ML_LABORFREIGABE_T11,
           Typ                      := 0,
           FBa                      := #xTmp,
           FBa2                     := #xTmp,
           Out                      := Q    259.3);

END_FUNCTION_BLOCK

FUNCTION_BLOCK FB 1111
TITLE =U011: Water Tank 11
FAMILY : BOTEC_F1
NAME : UniE
VERSION : 1.2


VAR_TEMP
  CIP : BOOL ;	//CIP active
  UNIM : BOOL ;	//Unit Not In Maintenance
  GenRel : BOOL ;	//general OK (emergency and maintenance OK)
  EStopOK : BOOL ;	//emergency OK
  UnitNo : INT ;	//unit number
  xTmp : BOOL ;	//Temporary Bool
  iTmp : INT ;	//Temporary INT
  rTmp : REAL ;	//Temporary REAL
  dTmp : DINT ;	//Temporary DINT (free for general use)
  RetValInt : INT ;	//return value
END_VAR
BEGIN
NETWORK
TITLE =General

      SET   ;
// Simulation ---------------------------------------------------------------
      A     DB1111.DBX 1357.7;
      CC    FB  1119; // "WT11Sim"
      A     DB1111.DBX   17.3;
      =     DB1111.DBX 1357.7; //Help bit for simulation

// get unit number ----------------------------------------------------------
      L     DB1110.DBW    0;
      T     #UnitNo;

// communication ------------------------------------------------------------
      UC    FB  1115; // WT11Com

NETWORK
TITLE =Sequence organisation

      CLR   ;
      =     M    122.2;

// CIP Counter
      CALL FC    29 (
           UnitNo                   := #UnitNo,
           Value                    := DB1115.DBD   54,
           Enable                   := TRUE,
           Down                     := FALSE,
           OriginDetect             := 0.000000e+000,
           MaxDiffPS                := 1.000000e+000,
           SFMRec                   := DB1111.Seq.SFM[15],
           ValueOld                 := DB1111.DBD 1418);

// sequencer ----------------------------------------------------------------
      A     DB1113.DBX   43.1;
      S     DB1113.DBX   97.3;

      CALL FC    40 (
           UnitNo                   := #UnitNo);

END_FUNCTION_BLOCK

FUNCTION_BLOCK FB 1120
TITLE =U012: Wassertank 12
FAMILY : BOTEC_F1
NAME : U012A
VERSION : 2.1


VAR_TEMP
  EStopOK : BOOL ;	//auxiliary flag
  CIP : BOOL ;	//CIP Program Selected
  xTmp : BOOL ;	//Temporary Bool(free for general use)
  DummyBool : BOOL ;	//Temporary Bool(free for general use)
  UnitNo : INT ;	//unit number
  UnitFB : INT ;	//unit expansion FB number
  rTmp : REAL ;	//Temporary REAL (free for general use)
  iTmp : INT ;	//Temporary INT (free for general use)
  DummyInt : INT ;	//Temporary INT (free for general use)
  dTmp : DINT ;	//Temporary DINT (free for general use)
END_VAR
BEGIN
NETWORK
TITLE =general

      CLR   ;
      =     #xTmp;
      =     #EStopOK;

      L     DB1120.DBW    0;
      T     #UnitNo;
      L     DB1120.DBW    2;
      T     #UnitFB;

NETWORK
TITLE =analog inputs

      NOP   0;
// LI_T12 AnI 001 Niveau Tank 12
      CALL FC    24 (
           UnitNo                   := #UnitNo,
           AnIRec                   := DB2123.LI_T12,
           ValPer                   := DB302.DBW   86);

NETWORK
TITLE =Universal value

      NOP   0;
// unv001 UnV 001 Process Status
      CALL FC    27 (
           UnitNo                   := #UnitNo,
           UnVRec                   := DB2125.unv001,
           ValExt                   := DB2125.DBD  234);

// unv002 UnV 002 Universal Value 02
      CALL FC    27 (
           UnitNo                   := #UnitNo,
           UnVRec                   := DB2125.unv002,
           ValExt                   := DB2125.DBD  362);

// unv003 UnV 003 Universal Value 03
      CALL FC    27 (
           UnitNo                   := #UnitNo,
           UnVRec                   := DB2125.unv003,
           ValExt                   := DB2125.DBD  490);

NETWORK
TITLE =special inputs

      NOP   0;
// LS_LLL_T12 SpI 001 LS- Tank 12
      CALL FC    14 (
           UnitNo                   := #UnitNo,
           SpIRec                   := DB2121.LS_LLL_T12,
           SpIBit                   := I     48.7);

// LS_HL_T12 SpI 002 LS+ Tank 12
      CALL FC    14 (
           UnitNo                   := #UnitNo,
           SpIRec                   := DB2121.LS_HL_T12,
           SpIBit                   := I     48.5);

// GOA_T12_ML SpI 003 Mannloch Tank 12
      CALL FC    14 (
           UnitNo                   := #UnitNo,
           SpIRec                   := DB2121.GOA_T12_ML,
           SpIBit                   := I     48.4);

// GOA_T12_VV SpI 004 Vacuumventil Tank 12
      CALL FC    14 (
           UnitNo                   := #UnitNo,
           SpIRec                   := DB2121.GOA_T12_VV,
           SpIBit                   := I     48.3);

// LS_LL_T12 SpI 005 LS/ Tank 12
      CALL FC    14 (
           UnitNo                   := #UnitNo,
           SpIRec                   := DB2121.LS_LL_T12,
           SpIBit                   := I     48.6);

// RM_NI_T12_K4_AUF SpI 006
      CALL FC    14 (
           UnitNo                   := #UnitNo,
           SpIRec                   := DB2121.RM_NI_T12_K4_AUF,
           SpIBit                   := I     48.1);

// RM_NI_T12_K4_ZU SpI 007
      CALL FC    14 (
           UnitNo                   := #UnitNo,
           SpIRec                   := DB2121.RM_NI_T12_K4_ZU,
           SpIBit                   := I     48.2);

// RM_NI_T12_K2 SpI 008
      CALL FC    14 (
           UnitNo                   := #UnitNo,
           SpIRec                   := DB2121.RM_NI_T12_K2,
           SpIBit                   := I    187.7);

// RM_NI_T12_K3 SpI 010
      CALL FC    14 (
           UnitNo                   := #UnitNo,
           SpIRec                   := DB2121.RM_NI_T12_K3,
           SpIBit                   := I     48.0);

// LABOR_FREIG_T12 SpI 011 SCHLUESSELSCHALTER LABOR
      CALL FC    14 (
           UnitNo                   := #UnitNo,
           SpIRec                   := DB2121.LABOR_FREIG_T12,
           SpIBit                   := I    259.4);

NETWORK
TITLE =messages

      NOP   0;
// msg001 Msg 001 Message 01
      CALL FC    16 (
           UnitNo                   := #UnitNo,
           MsgRec                   := DB2127.msg001,
           MsgBit                   := DB2127.DBX   82.7);

// msg002 Msg 002 Message 02
      CALL FC    16 (
           UnitNo                   := #UnitNo,
           MsgRec                   := DB2127.msg002,
           MsgBit                   := DB2127.DBX  142.7);

NETWORK
TITLE =unit supply

      UC    FB [#UnitFB];

NETWORK
TITLE =T12_A10
// Act 005
// Box           : Ventilinsel 2
// Input address : I317.3
// Output address: Q317.3
      CALL FC    70 (
           UnitNo                   := #UnitNo,
           ActRec                   := DB2120.T12_A10,
           Typ                      := 1,
           FBa                      := #xTmp,
           FBa2                     := I    317.3,
           Out                      := Q    317.3);

NETWORK
TITLE =T12_A9
// Act 006
// Box           : Ventilinsel 2
// Input address : I319.3
// Output address: Q319.3
      CALL FC    70 (
           UnitNo                   := #UnitNo,
           ActRec                   := DB2120.T12_A9,
           Typ                      := 1,
           FBa                      := #xTmp,
           FBa2                     := I    319.3,
           Out                      := Q    319.3);

NETWORK
TITLE =T12_A12
// Act 007
// Box           : Ventilinsel 2
// Input address : I321.3
// Output address: Q321.3
      CALL FC    70 (
           UnitNo                   := #UnitNo,
           ActRec                   := DB2120.T12_A12,
           Typ                      := 1,
           FBa                      := #xTmp,
           FBa2                     := I    321.3,
           Out                      := Q    321.3);

NETWORK
TITLE =T12_A7
// Act 008
// Box           : Ventilinsel 2
// Input address : I323.3
// Output address: Q323.3
      CALL FC    70 (
           UnitNo                   := #UnitNo,
           ActRec                   := DB2120.T12_A7,
           Typ                      := 1,
           FBa                      := #xTmp,
           FBa2                     := I    323.3,
           Out                      := Q    323.3);

NETWORK
TITLE =T12_A8
// Act 009
// Box           : Ventilinsel 3
// Input address : I325.3
// Output address: Q325.3
      CALL FC    70 (
           UnitNo                   := #UnitNo,
           ActRec                   := DB2120.T12_A8,
           Typ                      := 1,
           FBa                      := #xTmp,
           FBa2                     := I    325.3,
           Out                      := Q    325.3);

NETWORK
TITLE =T12_A5
// Act 010
// Box           : Ventilinsel 3
// Input address : I327.3
// Output address: Q327.3
      CALL FC    70 (
           UnitNo                   := #UnitNo,
           ActRec                   := DB2120.T12_A5,
           Typ                      := 1,
           FBa                      := #xTmp,
           FBa2                     := I    327.3,
           Out                      := Q    327.3);

NETWORK
TITLE =T12_A11
// Act 011
// Box           : Ventilinsel 3
// Input address : I329.3
// Output address: Q329.3
      CALL FC    70 (
           UnitNo                   := #UnitNo,
           ActRec                   := DB2120.T12_A11,
           Typ                      := 1,
           FBa                      := #xTmp,
           FBa2                     := I    329.3,
           Out                      := Q    329.3);

NETWORK
TITLE =T12_A14
// Act 012
// Box           : Ventilinsel 4
// Input address : I331.3
// Output address: Q331.3
      CALL FC    70 (
           UnitNo                   := #UnitNo,
           ActRec                   := DB2120.T12_A14,
           Typ                      := 1,
           FBa                      := #xTmp,
           FBa2                     := I    331.3,
           Out                      := Q    331.3);

NETWORK
TITLE =T12_A15
// Act 013
// Box           : Ventilinsel 4
// Input address : I333.3
// Output address: Q333.3
      CALL FC    70 (
           UnitNo                   := #UnitNo,
           ActRec                   := DB2120.T12_A15,
           Typ                      := 0,
           FBa                      := #xTmp,
           FBa2                     := I    333.3,
           Out                      := Q    333.3);

NETWORK
TITLE =T12_RR1
// Act 014
// Box           : Ventilinsel 4
// Input address : I335.3
// Output address: Q335.3
      CALL FC    70 (
           UnitNo                   := #UnitNo,
           ActRec                   := DB2120.T12_RR1,
           Typ                      := 1,
           FBa                      := #xTmp,
           FBa2                     := I    335.3,
           Out                      := Q    335.3);

NETWORK
TITLE =RV1_T12
// Act 015
// Box           : Ventilinsel 1
// Input address : I9.2
// Output address: Q9.2
      CALL FC    70 (
           UnitNo                   := #UnitNo,
           ActRec                   := DB2120.RV1_T12,
           Typ                      := 1,
           FBa                      := #xTmp,
           FBa2                     := I      9.2,
           Out                      := Q      9.2);

NETWORK
TITLE =B6F_T12
// Act 016
// Box           : Ventilinsel 1
// Input address : I9.3
// Output address: Q9.3
      CALL FC    70 (
           UnitNo                   := #UnitNo,
           ActRec                   := DB2120.B6F_T12,
           Typ                      := 1,
           FBa                      := #xTmp,
           FBa2                     := I      9.3,
           Out                      := Q      9.3);

NETWORK
TITLE =H6F_T12
// Act 017
// Box           : Ventilinsel 1
// Input address : I9.4
// Output address: Q9.4
      CALL FC    70 (
           UnitNo                   := #UnitNo,
           ActRec                   := DB2120.H6F_T12,
           Typ                      := 1,
           FBa                      := #xTmp,
           FBa2                     := I      9.4,
           Out                      := Q      9.4);

NETWORK
TITLE =J6F_T12
// Act 018
// Box           : Ventilinsel 1
// Input address : I9.5
// Output address: Q9.5
      CALL FC    70 (
           UnitNo                   := #UnitNo,
           ActRec                   := DB2120.J6F_T12,
           Typ                      := 1,
           FBa                      := #xTmp,
           FBa2                     := I      9.5,
           Out                      := Q      9.5);

NETWORK
TITLE =L6F_T12
// Act 019
// Box           : Ventilinsel 1
// Input address : I9.6
// Output address: Q9.6
      CALL FC    70 (
           UnitNo                   := #UnitNo,
           ActRec                   := DB2120.L6F_T12,
           Typ                      := 1,
           FBa                      := #xTmp,
           FBa2                     := I      9.6,
           Out                      := Q      9.6);

NETWORK
TITLE =D6_T12
// Act 020
// Box           : Ventilinsel 1
// Input address : I9.7
// Output address: Q9.7
      CALL FC    70 (
           UnitNo                   := #UnitNo,
           ActRec                   := DB2120.D6_T12,
           Typ                      := 1,
           FBa                      := #xTmp,
           FBa2                     := I      9.7,
           Out                      := Q      9.7);

NETWORK
TITLE =B6_T12
// Act 021
// Box           : Ventilinsel 1
// Input address : I10.0
// Output address: Q10.0
      CALL FC    70 (
           UnitNo                   := #UnitNo,
           ActRec                   := DB2120.B6_T12,
           Typ                      := 1,
           FBa                      := #xTmp,
           FBa2                     := I     10.0,
           Out                      := Q     10.0);

NETWORK
TITLE =A_T12
// Act 022
// Box           : Ventilinsel 1
// Input address : I10.1
// Output address: Q10.1
      CALL FC    70 (
           UnitNo                   := #UnitNo,
           ActRec                   := DB2120.A_T12,
           Typ                      := 1,
           FBa                      := #xTmp,
           FBa2                     := I     10.1,
           Out                      := Q     10.1);

NETWORK
TITLE =B_T12
// Act 023
// Box           : Ventilinsel 1
// Input address : I10.2
// Output address: Q10.2
      CALL FC    70 (
           UnitNo                   := #UnitNo,
           ActRec                   := DB2120.B_T12,
           Typ                      := 1,
           FBa                      := #xTmp,
           FBa2                     := I     10.2,
           Out                      := Q     10.2);

NETWORK
TITLE =CF_T12
// Act 024
// Box           : Ventilinsel 1
// Input address : I17.5
// Output address: Q17.5
      CALL FC    70 (
           UnitNo                   := #UnitNo,
           ActRec                   := DB2120.CF_T12,
           Typ                      := 1,
           FBa                      := #xTmp,
           FBa2                     := I     17.5,
           Out                      := Q     17.5);

NETWORK
TITLE =C_T12
// Act 025
// Box           : VS2-BB
// Input address : I311.5
// Output address: Q311.5
      CALL FC    70 (
           UnitNo                   := #UnitNo,
           ActRec                   := DB2120.C_T12,
           Typ                      := 1,
           FBa                      := #xTmp,
           FBa2                     := I    311.5,
           Out                      := Q    311.5);

NETWORK
TITLE =VVT12  Vacuumventil Tank 12
// Act 028
// Box           : VST1-9
// Output address: Q160.1
      CALL FC    70 (
           UnitNo                   := #UnitNo,
           ActRec                   := DB2120.VVT12,
           Typ                      := 0,
           FBa                      := #xTmp,
           FBa2                     := #xTmp,
           Out                      := Q    160.1);

NETWORK
TITLE =VR_T12
// Act 029
// Box           : Ventilinsel 1
// Output address: Q10.3
      CALL FC    70 (
           UnitNo                   := #UnitNo,
           ActRec                   := DB2120.VR_T12,
           Typ                      := 0,
           FBa                      := #xTmp,
           FBa2                     := #xTmp,
           Out                      := Q     10.3);

NETWORK
TITLE =ML_LABORFREIGABE_T12
// Act 031
// Box           : LT-CIP
// Output address: Q259.4
      CALL FC    70 (
           UnitNo                   := #UnitNo,
           ActRec                   := DB2120.ML_LABORFREIGABE_T12,
           Typ                      := 0,
           FBa                      := #xTmp,
           FBa2                     := #xTmp,
           Out                      := Q    259.4);

END_FUNCTION_BLOCK

FUNCTION_BLOCK FB 1121
TITLE =U012: Water Tank 12
FAMILY : BOTEC_F1
NAME : UniE
VERSION : 1.2


VAR_TEMP
  CIP : BOOL ;	//CIP active
  UNIM : BOOL ;	//Unit Not In Maintenance
  GenRel : BOOL ;	//general OK (emergency and maintenance OK)
  EStopOK : BOOL ;	//emergency OK
  UnitNo : INT ;	//unit number
  xTmp : BOOL ;	//Temporary Bool
  iTmp : INT ;	//Temporary INT
  rTmp : REAL ;	//Temporary REAL
  dTmp : DINT ;	//Temporary DINT (free for general use)
  RetValInt : INT ;	//return value
END_VAR
BEGIN
NETWORK
TITLE =General

// Simulation ---------------------------------------------------------------
      A     DB1121.DBX 1357.7;
      CC    FB  1129; // "WT12Sim"
      A     DB1121.DBX   17.3;
      =     DB1121.DBX 1357.7; //Help bit for simulation

